PROGRAM Main
VAR
	KWP_SP_AC_NC_0: KWP_SP_AC_NC;
	VD_0: VD;
	KD_0: KD;
	Kreis_3KO_0: Kreis_3KO;
	HWP_SP_0: HWP_SP;
	Zusatzheizung_0: Zusatzheizung;
	Zirk_Pumpe_0: Zirk_Pumpe;
	TWW_SP_0: TWW_SP;
	Init_0: Init;
	IOs_0: IOs;
	AI_to_Druck_0: AI_to_Druck;
	AI_to_Druck_1: AI_to_Druck;
END_VAR
VAR PERSISTENT
	dut_Liste:SW_Struct;
END_VAR

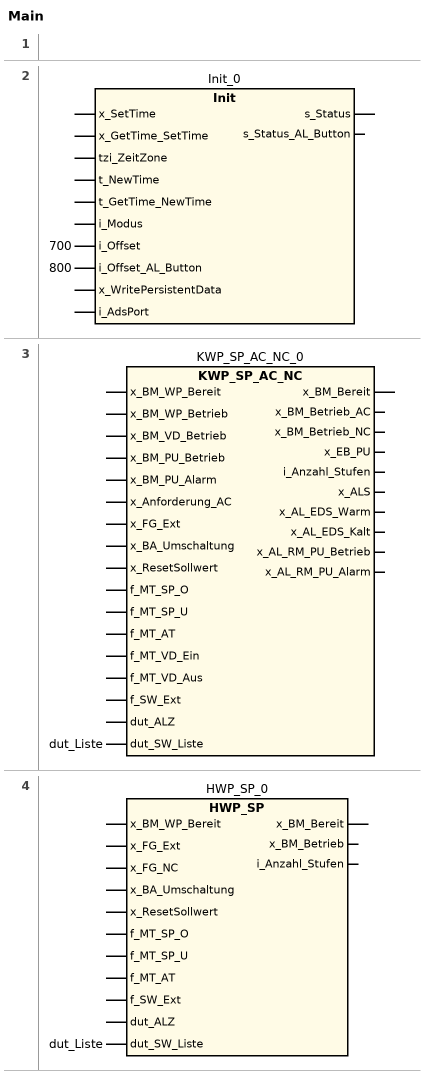
// NETWORK 1

// NETWORK 2
Init_0(i_Offset := 700, i_Offset_AL_Button := 800); // Init

// NETWORK 3
KWP_SP_AC_NC_0(dut_SW_Liste := dut_Liste); // KWP_SP_AC_NC

// NETWORK 4
HWP_SP_0(dut_SW_Liste := dut_Liste); // HWP_SP

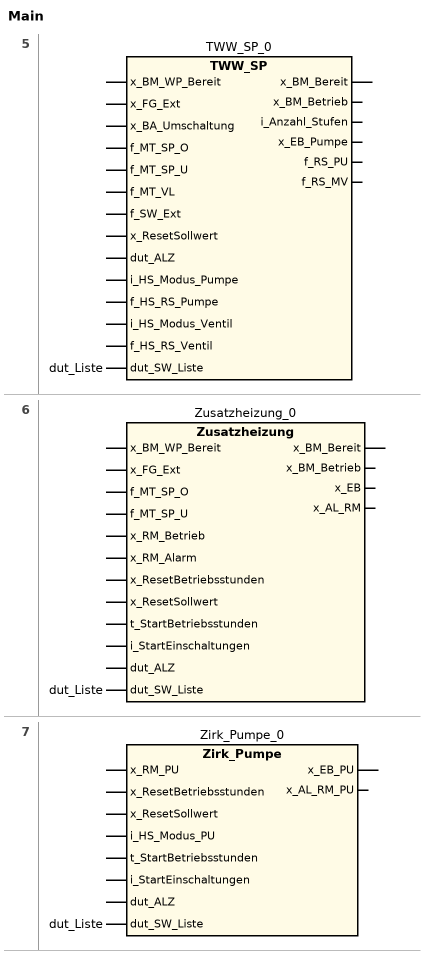
// NETWORK 5
TWW_SP_0(dut_SW_Liste := dut_Liste); // TWW_SP

// NETWORK 6
Zusatzheizung_0(dut_SW_Liste := dut_Liste); // Zusatzheizung

// NETWORK 7
Zirk_Pumpe_0(dut_SW_Liste := dut_Liste); // Zirk_Pumpe

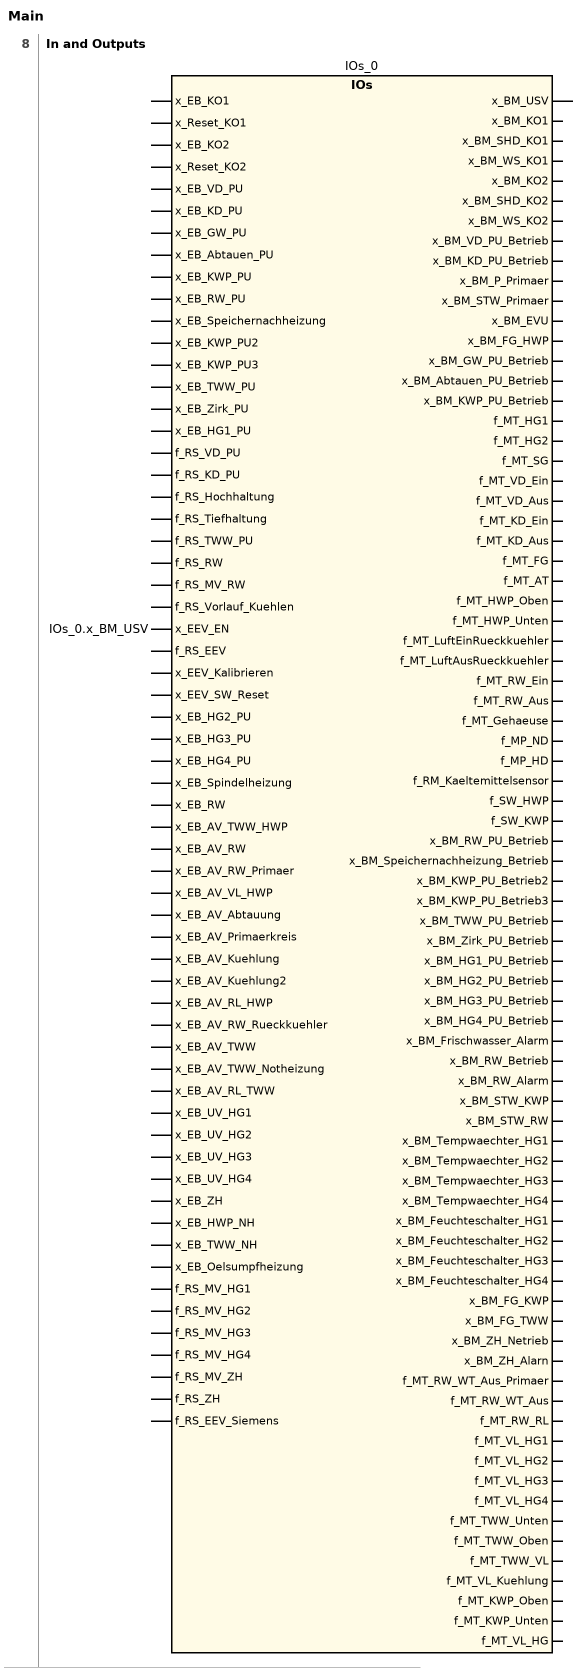
// NETWORK 8: In and Outputs
IOs_0(x_EEV_EN := IOs_0.x_BM_USV); // IOs

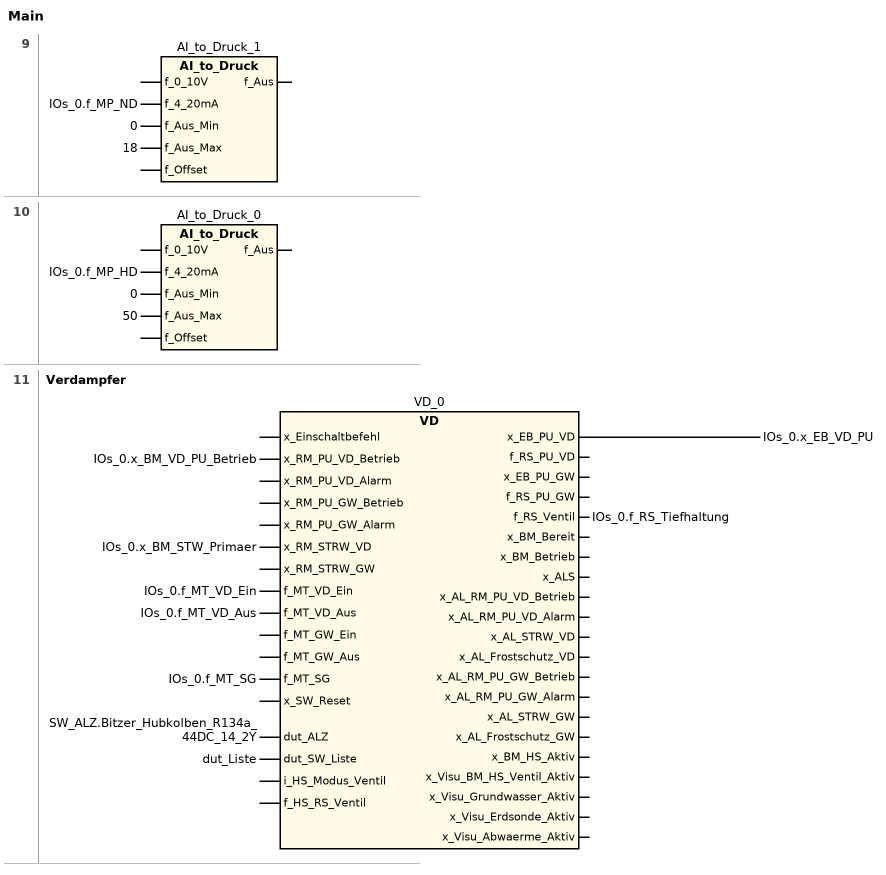
// NETWORK 9
AI_to_Druck_1(f_4_20mA := IOs_0.f_MP_ND, f_Aus_Min := 0, f_Aus_Max := 18); // AI_to_Druck

// NETWORK 10
AI_to_Druck_0(f_4_20mA := IOs_0.f_MP_HD, f_Aus_Min := 0, f_Aus_Max := 50); // AI_to_Druck

// NETWORK 11: Verdampfer
VD_0(
    x_RM_PU_VD_Betrieb := IOs_0.x_BM_VD_PU_Betrieb,
    x_RM_STRW_VD := IOs_0.x_BM_STW_Primaer,
    f_MT_VD_Ein := IOs_0.f_MT_VD_Ein,
    f_MT_VD_Aus := IOs_0.f_MT_VD_Aus,
    f_MT_SG := IOs_0.f_MT_SG,
    dut_ALZ := SW_ALZ.Bitzer_Hubkolben_R134a_44DC_14_2Y,
    dut_SW_Liste := dut_Liste,
    f_RS_Ventil => IOs_0.f_RS_Tiefhaltung); // VD
IOs_0.x_EB_VD_PU := VD_0.x_EB_PU_VD;

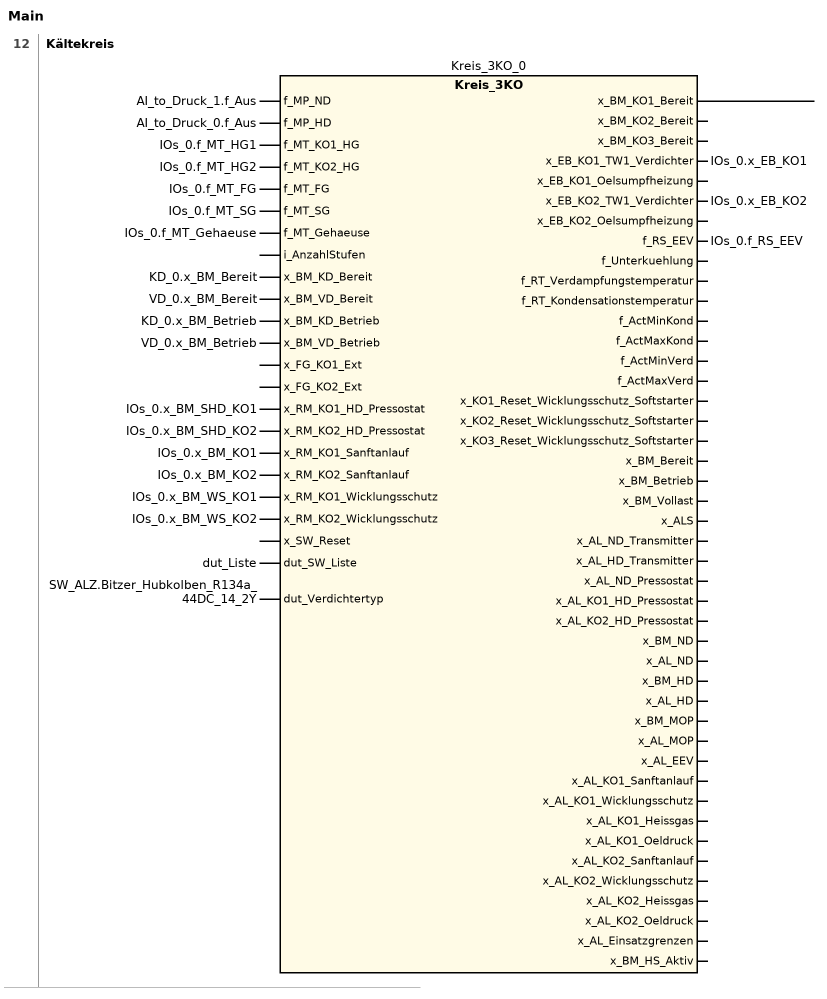
// NETWORK 12: Kältekreis
Kreis_3KO_0(
    f_MP_ND := AI_to_Druck_1.f_Aus,
    f_MP_HD := AI_to_Druck_0.f_Aus,
    f_MT_KO1_HG := IOs_0.f_MT_HG1,
    f_MT_KO2_HG := IOs_0.f_MT_HG2,
    f_MT_FG := IOs_0.f_MT_FG,
    f_MT_SG := IOs_0.f_MT_SG,
    f_MT_Gehaeuse := IOs_0.f_MT_Gehaeuse,
    x_BM_KD_Bereit := KD_0.x_BM_Bereit,
    x_BM_VD_Bereit := VD_0.x_BM_Bereit,
    x_BM_KD_Betrieb := KD_0.x_BM_Betrieb,
    x_BM_VD_Betrieb := VD_0.x_BM_Betrieb,
    x_RM_KO1_HD_Pressostat := IOs_0.x_BM_SHD_KO1,
    x_RM_KO2_HD_Pressostat := IOs_0.x_BM_SHD_KO2,
    x_RM_KO1_Sanftanlauf := IOs_0.x_BM_KO1,
    x_RM_KO2_Sanftanlauf := IOs_0.x_BM_KO2,
    x_RM_KO1_Wicklungsschutz := IOs_0.x_BM_WS_KO1,
    x_RM_KO2_Wicklungsschutz := IOs_0.x_BM_WS_KO2,
    dut_SW_Liste := dut_Liste,
    dut_Verdichtertyp := SW_ALZ.Bitzer_Hubkolben_R134a_44DC_14_2Y,
    x_EB_KO1_TW1_Verdichter => IOs_0.x_EB_KO1,
    x_EB_KO2_TW1_Verdichter => IOs_0.x_EB_KO2,
    f_RS_EEV => IOs_0.f_RS_EEV); // Kreis_3KO

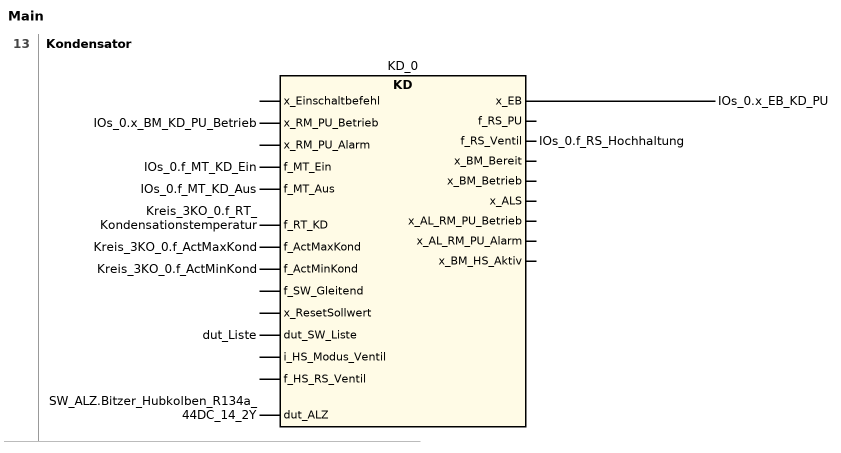
// NETWORK 13: Kondensator
KD_0(
    x_RM_PU_Betrieb := IOs_0.x_BM_KD_PU_Betrieb,
    f_MT_Ein := IOs_0.f_MT_KD_Ein,
    f_MT_Aus := IOs_0.f_MT_KD_Aus,
    f_RT_KD := Kreis_3KO_0.f_RT_Kondensationstemperatur,
    f_ActMaxKond := Kreis_3KO_0.f_ActMaxKond,
    f_ActMinKond := Kreis_3KO_0.f_ActMinKond,
    dut_SW_Liste := dut_Liste,
    dut_ALZ := SW_ALZ.Bitzer_Hubkolben_R134a_44DC_14_2Y,
    f_RS_Ventil => IOs_0.f_RS_Hochhaltung); // KD
IOs_0.x_EB_KD_PU := KD_0.x_EB;

END_PROGRAM

(* stored: Version 1.1.0.1, ProductVersion 3.1.4022.6
   POU Main: Id {bcf30e2d-0792-4814-9d4c-a58e87c7eb2d}, SpecialFunc None *)
